PROGRAM MAIN
VAR
END_VAR

Door_Control();
Light_Control();

END_PROGRAM

(* stored: Version 1.1.0.1, ProductVersion 3.1.4024.15
   POU MAIN: Id {9a27226a-4db9-492c-aff9-e3c1f67a97bd}, SpecialFunc None *)
